FUNCTION_BLOCK Scale_Int
TITLE = 'Scale an Integer Input Value'

VAR_INPUT
    ScaleFromMin : INT;   // Minimum value of input range
    ScaleFromMax : INT;   // Maximum value of input range
    ScaleToMin   : INT;   // Minimum value of output range
    ScaleToMax   : INT;   // Maximum value of output range
    PV           : INT;   // Input value to be scaled
END_VAR

VAR_OUTPUT
    ScaledPV     : INT;   // Output value scaled to output range
END_VAR

VAR
    ScaleFactor  : INT;   // Scale factor to map input range to output range
    Offset       : INT;   // Offset to add to scaled value to get output in output range
END_VAR

// Calculate scale factor and offset
ScaleFactor := (ScaleToMax - ScaleToMin) / (ScaleFromMax - ScaleFromMin);
Offset := ScaleToMin - ScaleFactor * ScaleFromMin;

// Scale input value to output range
ScaledPV := PV * ScaleFactor + Offset;

END_FUNCTION_BLOCK
